Fanuc KAREL source: kt00037.KL

PROGRAM KT00037
%STACKSIZE=65535
%PRIORITY=65535
%NOLOCKGROUP
VAR
I1 : INTEGER
OUT : INTEGER
-- UNRESOLVED DECLARATIONS (source type spelling not recovered)
-- Y2 : ARRAY[2] OF TYPE_0x0018 (type_u16=0x2018)
BEGIN
I1=2
Y2[1]=3
-- UNRESOLVED_PC line 10 opcodes [21 22 9D 33 B1 53 23] marker_code=35
END KT00037
